RoboDK station: tx2-40-hb.rdk

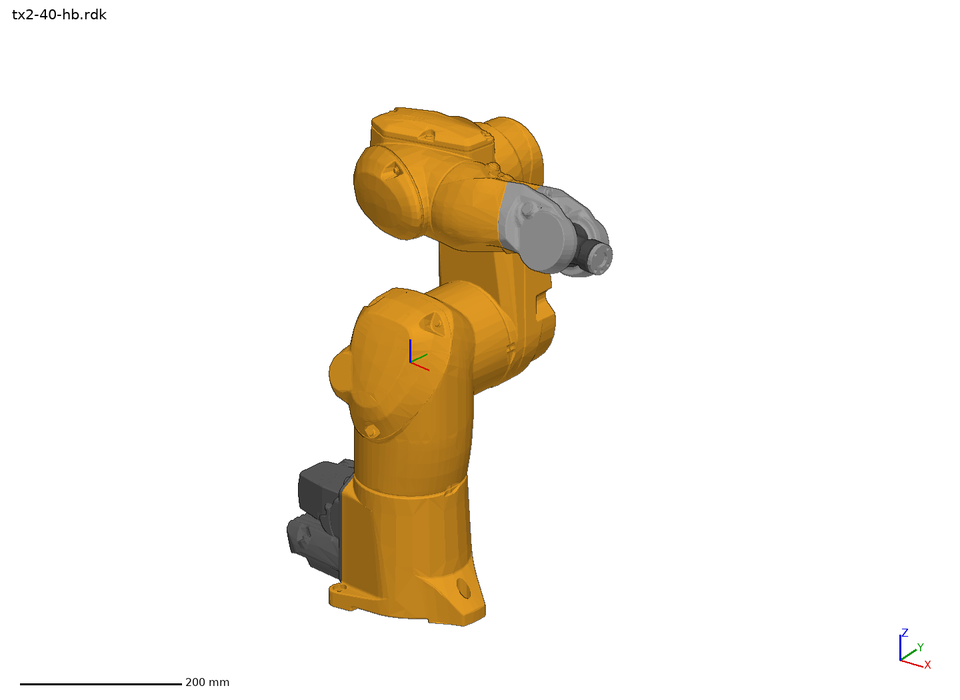
[picture v0: the station drawn from its stored meshes, robots at their saved joint values, targets as dots, program paths as lines]
Station tx2-40-hb (saved by RoboDK 5.4.0). Poses are relative to the parent item; angles as X-Y-Z fixed-axis rotations.
  - frame Staubli TX2-40 Base at (0, 0, 320) mm, rotated rx 0 ry 0 rz -7.68 deg
    - robot Staubli TX2-40: 6 axes, payload 1.7 kg, reach 515 mm, repeatability 0.02 mm, weight 29 kg
        modified DH rows (alpha deg, a mm, theta deg, d mm): 0, 0, 0, 320; -90, 0, -90, 35; 0, 225, -90, 0; -90, 0, 0, 225; 90, 0, 0, 0; -90, 0, 180, 65
        base shift (0, 0, -320) mm
        joint limits [-180, -125, -138, -270, -120, -270] to [180, 125, 138, 270, 133.5, 270]; home [0, 0, 90, 0, 0, 0]; saved at [0, 0, 90, -24.341, 0, 24.341]
